{attribute addProperty BoxType "EL3702-0000-0002"}
{attribute addProperty Id "Ch1_CycleCountAT %I*Ch1_CycleCount_2F207C3C1620Ch1_SampleAT %I*ARRAY[0..9] OF Ch1_Sample_37C07C83160200Ch2_CycleCountAT %I*Ch2_CycleCount_7D759C541620Ch2_SampleAT %I*ARRAY[0..9] OF Ch2_Sample_29ECE468160200WcStateAT %I*WcState_98A4DF7520.250InfoDataAT %I*InfoData_7231B2DD80100"}
{attribute addProperty CRC "1838895957"}
{attribute addProperty SizeInBites "434"}
{attribute addProperty SizeInBytes "54.25"}
TYPE EL3702_72DB3B79 :
STRUCT
	{attribute addProperty Name "Ch1_CycleCount"}
	Ch1_CycleCount : Ch1_CycleCount_2F207C3C;
	{attribute addProperty Name "Ch1_Sample"}
	Ch1_Sample : ARRAY[0..9] OF Ch1_Sample_37C07C83;
	{attribute addProperty Name "Ch2_CycleCount"}
	Ch2_CycleCount : Ch2_CycleCount_7D759C54;
	{attribute addProperty Name "Ch2_Sample"}
	Ch2_Sample : ARRAY[0..9] OF Ch2_Sample_29ECE468;
	{attribute addProperty Name "WcState"}
	WcState : WcState_98A4DF75;
	{attribute addProperty Name "InfoData"}
	InfoData : InfoData_7231B2DD;
END_STRUCT
END_TYPE

(* stored: Version 1.2.0.0, ProductVersion 3.1.4024.9
   DUT EL3702_72DB3B79: Id {bebd0b3e-3d6f-461f-882e-286b682d7794} *)
